// TIA Portal V16 export
// export: Created 2021-08-16T21:06:41.371237Z, ExportSetting WithDefaults, DisplayName Totally Integrated Automation Portal, DisplayVersion V16, DisplayName TIA Portal Version Control Interface, DisplayVersion V16, DisplayName TIA Portal Openness, DisplayVersion V16, DisplayName STEP 7 Professional, DisplayVersion V16, DisplayName STEP 7 Safety, DisplayVersion V16, DisplayName WinCC Advanced, DisplayVersion V16
ORGANIZATION_BLOCK "Main"   // OB1, LAD, ProgramCycle
TITLE = "Main Program Sweep (Cycle)"
{ S7_Optimized_Access := 'TRUE' }
VERSION : 0.1
// stored: AutoNumber true, IsIECCheckEnabled false, SetENOAutomatically false
   VAR_INPUT
      Initial_Call : Bool;   // Initial call of this OB
      Remanence : Bool;   // =True, if remanent data are available
   END_VAR
   VAR CONSTANT
      start : Bool;
   END_VAR
BEGIN

REGION Network 1: Spustenie a zastavenie automatického režimu
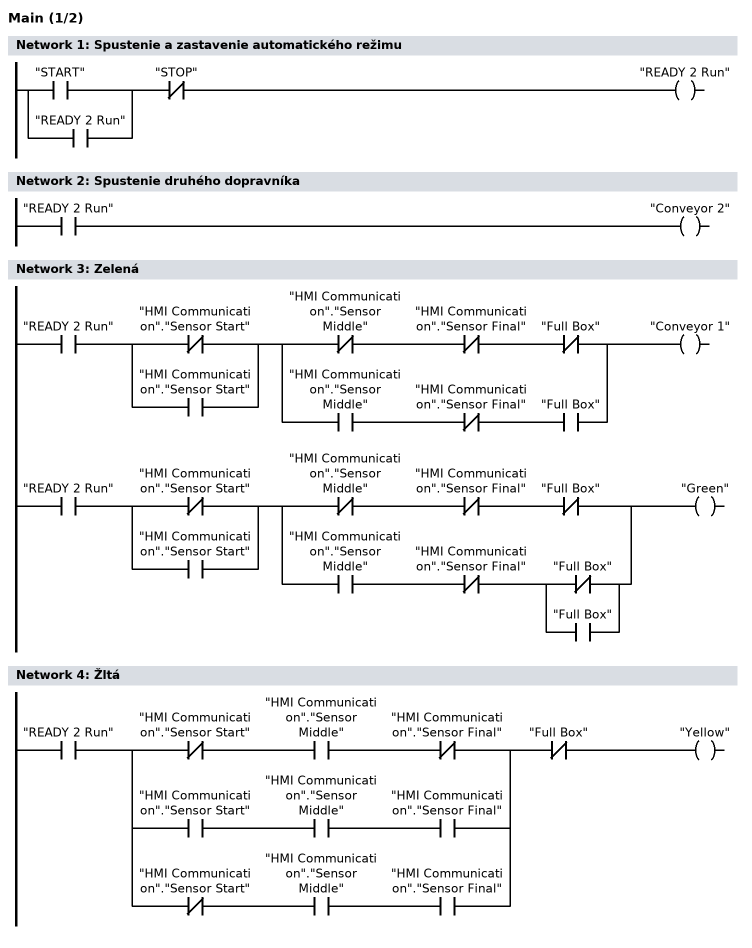
   RUNG wire#powerrail
      Contact( "START" )
      wire#w1
      I_Contact( "STOP" )
      Coil( "READY 2 Run" )
   END_RUNG
   RUNG wire#powerrail
      Contact( "READY 2 Run" )
   END_RUNG wire#w1
   // the same network as SCL:
   "READY 2 Run" := ("START" OR "READY 2 Run") AND NOT "STOP";
END_REGION

REGION Network 2: Spustenie druhého dopravníka
   RUNG wire#powerrail
      Contact( "READY 2 Run" )
      Coil( "Conveyor 2" )
   END_RUNG
   // the same network as SCL:
   "Conveyor 2" := "READY 2 Run";
END_REGION

REGION Network 3: Zelená
   RUNG wire#powerrail
      Contact( "READY 2 Run" )
      wire#w1
      I_Contact( "HMI Communication"."Sensor Start" )
      wire#w2
      I_Contact( "HMI Communication"."Sensor Middle" )
      I_Contact( "HMI Communication"."Sensor Final" )
      I_Contact( "Full Box" )
      wire#w3
      Coil( "Conveyor 1" )
   END_RUNG
   RUNG wire#w1
      Contact( "HMI Communication"."Sensor Start" )
   END_RUNG wire#w2
   RUNG wire#w2
      Contact( "HMI Communication"."Sensor Middle" )
      I_Contact( "HMI Communication"."Sensor Final" )
      Contact( "Full Box" )
   END_RUNG wire#w3
   RUNG wire#powerrail
      Contact( "READY 2 Run" )
      wire#w4
      I_Contact( "HMI Communication"."Sensor Start" )
      wire#w5
      I_Contact( "HMI Communication"."Sensor Middle" )
      I_Contact( "HMI Communication"."Sensor Final" )
      I_Contact( "Full Box" )
      wire#w6
      Coil( "Green" )
   END_RUNG
   RUNG wire#w4
      Contact( "HMI Communication"."Sensor Start" )
   END_RUNG wire#w5
   RUNG wire#w5
      Contact( "HMI Communication"."Sensor Middle" )
      I_Contact( "HMI Communication"."Sensor Final" )
      wire#w7
      I_Contact( "Full Box" )
   END_RUNG wire#w6
   RUNG wire#w7
      Contact( "Full Box" )
   END_RUNG wire#w6
   // the same network as SCL:
   "Conveyor 1" := "READY 2 Run" AND (NOT "HMI Communication"."Sensor Start" OR "HMI Communication"."Sensor Start") AND ((NOT "HMI Communication"."Sensor Middle" AND NOT "HMI Communication"."Sensor Final" AND NOT "Full Box") OR ("HMI Communication"."Sensor Middle" AND NOT "HMI Communication"."Sensor Final" AND "Full Box"));
   "Green" := "READY 2 Run" AND (NOT "HMI Communication"."Sensor Start" OR "HMI Communication"."Sensor Start") AND ((NOT "HMI Communication"."Sensor Middle" AND NOT "HMI Communication"."Sensor Final" AND NOT "Full Box") OR ("HMI Communication"."Sensor Middle" AND NOT "HMI Communication"."Sensor Final" AND (NOT "Full Box" OR "Full Box")));
END_REGION

REGION Network 4: Žltá
   RUNG wire#powerrail
      Contact( "READY 2 Run" )
      wire#w1
      I_Contact( "HMI Communication"."Sensor Start" )
      Contact( "HMI Communication"."Sensor Middle" )
      I_Contact( "HMI Communication"."Sensor Final" )
      wire#w2
      I_Contact( "Full Box" )
      Coil( "Yellow" )
   END_RUNG
   RUNG wire#w1
      Contact( "HMI Communication"."Sensor Start" )
      Contact( "HMI Communication"."Sensor Middle" )
      Contact( "HMI Communication"."Sensor Final" )
   END_RUNG wire#w2
   RUNG wire#w1
      I_Contact( "HMI Communication"."Sensor Start" )
      Contact( "HMI Communication"."Sensor Middle" )
      Contact( "HMI Communication"."Sensor Final" )
   END_RUNG wire#w2
   // the same network as SCL:
   "Yellow" := "READY 2 Run" AND ((NOT "HMI Communication"."Sensor Start" AND "HMI Communication"."Sensor Middle" AND NOT "HMI Communication"."Sensor Final") OR ("HMI Communication"."Sensor Start" AND "HMI Communication"."Sensor Middle" AND "HMI Communication"."Sensor Final") OR (NOT "HMI Communication"."Sensor Start" AND "HMI Communication"."Sensor Middle" AND "HMI Communication"."Sensor Final")) AND NOT "Full Box";
END_REGION

REGION Network 5: Červená
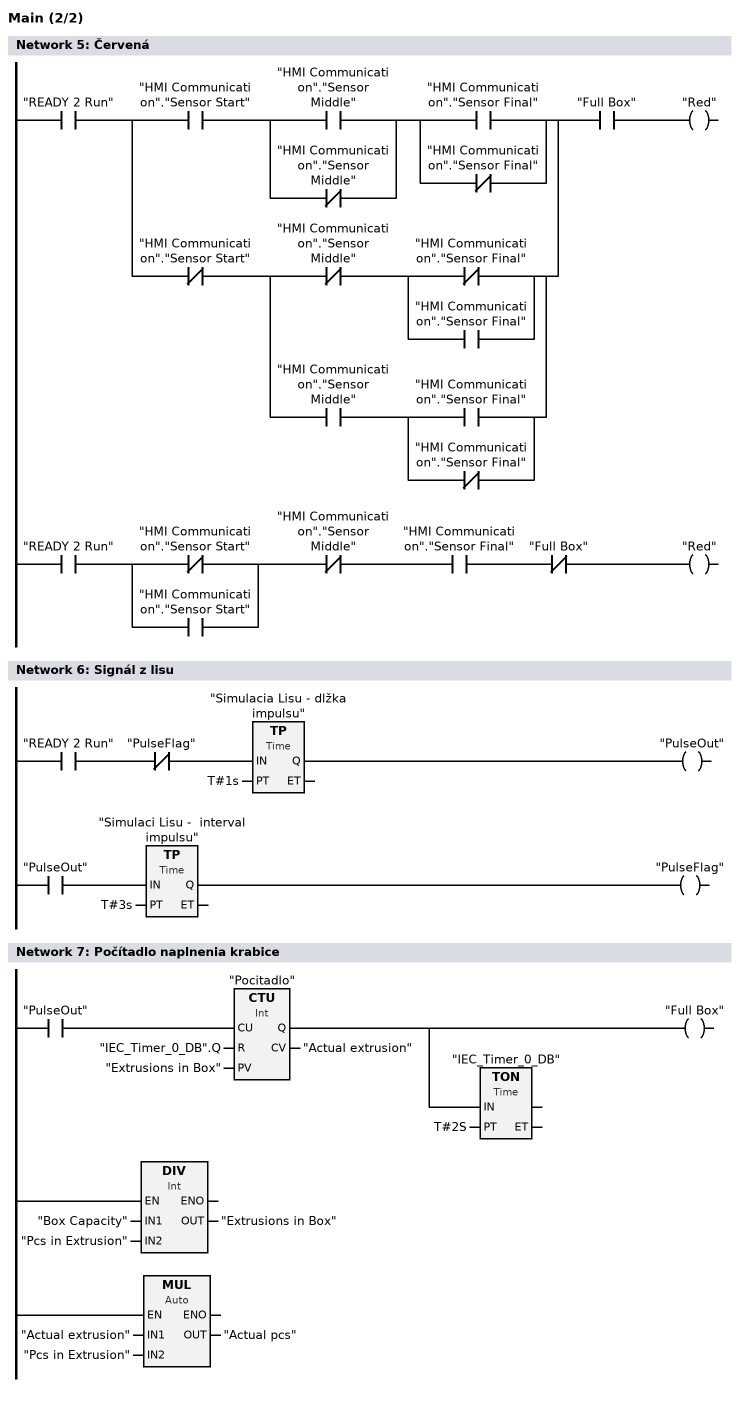
   RUNG wire#powerrail
      Contact( "READY 2 Run" )
      wire#w1
      Contact( "HMI Communication"."Sensor Start" )
      wire#w2
      Contact( "HMI Communication"."Sensor Middle" )
      wire#w3
      Contact( "HMI Communication"."Sensor Final" )
      wire#w4
      Contact( "Full Box" )
      Coil( "Red" )
   END_RUNG
   RUNG wire#w2
      I_Contact( "HMI Communication"."Sensor Middle" )
   END_RUNG wire#w3
   RUNG wire#w3
      I_Contact( "HMI Communication"."Sensor Final" )
   END_RUNG wire#w4
   RUNG wire#w1
      I_Contact( "HMI Communication"."Sensor Start" )
      wire#w5
      I_Contact( "HMI Communication"."Sensor Middle" )
      wire#w6
      I_Contact( "HMI Communication"."Sensor Final" )
   END_RUNG wire#w4
   RUNG wire#w6
      Contact( "HMI Communication"."Sensor Final" )
   END_RUNG wire#w4
   RUNG wire#w5
      Contact( "HMI Communication"."Sensor Middle" )
      wire#w7
      Contact( "HMI Communication"."Sensor Final" )
   END_RUNG wire#w4
   RUNG wire#w7
      I_Contact( "HMI Communication"."Sensor Final" )
   END_RUNG wire#w4
   RUNG wire#powerrail
      Contact( "READY 2 Run" )
      wire#w8
      I_Contact( "HMI Communication"."Sensor Start" )
      wire#w9
      I_Contact( "HMI Communication"."Sensor Middle" )
      Contact( "HMI Communication"."Sensor Final" )
      I_Contact( "Full Box" )
      Coil( "Red" )
   END_RUNG
   RUNG wire#w8
      Contact( "HMI Communication"."Sensor Start" )
   END_RUNG wire#w9
   // the same network as SCL:
   "Red" := "READY 2 Run" AND (("HMI Communication"."Sensor Start" AND ("HMI Communication"."Sensor Middle" OR NOT "HMI Communication"."Sensor Middle") AND ("HMI Communication"."Sensor Final" OR NOT "HMI Communication"."Sensor Final")) OR (NOT "HMI Communication"."Sensor Start" AND ((NOT "HMI Communication"."Sensor Middle" AND (NOT "HMI Communication"."Sensor Final" OR "HMI Communication"."Sensor Final")) OR ("HMI Communication"."Sensor Middle" AND ("HMI Communication"."Sensor Final" OR NOT "HMI Communication"."Sensor Final"))))) AND "Full Box";
   "Red" := "READY 2 Run" AND (NOT "HMI Communication"."Sensor Start" OR "HMI Communication"."Sensor Start") AND NOT "HMI Communication"."Sensor Middle" AND "HMI Communication"."Sensor Final" AND NOT "Full Box";
END_REGION

REGION Network 6: Signál z lisu
   RUNG wire#powerrail
      Contact( "READY 2 Run" )
      I_Contact( "PulseFlag" )
      { S7_Templates := "time_type := Time" } "Simulacia Lisu - dlžka impulsu".TP(pt := T#1s, et =>)
      Coil( "PulseOut" )
   END_RUNG
   RUNG wire#powerrail
      Contact( "PulseOut" )
      { S7_Templates := "time_type := Time" } "Simulaci Lisu -  interval impulsu".TP(pt := T#3s, et =>)
      Coil( "PulseFlag" )
   END_RUNG
   // the same network as SCL:
   "Simulacia Lisu - dlžka impulsu".TP(IN := "READY 2 Run" AND NOT "PulseFlag", PT := T#1s);
   "PulseOut" := "Simulacia Lisu - dlžka impulsu".Q;
   "Simulaci Lisu -  interval impulsu".TP(IN := "PulseOut", PT := T#3s);
   "PulseFlag" := "Simulaci Lisu -  interval impulsu".Q;
END_REGION

REGION Network 7: Počítadlo naplnenia krabice
   RUNG wire#powerrail
      Contact( "PulseOut" )
      { S7_Templates := "value_type := Int" } "Pocitadlo".CTU(r := "IEC_Timer_0_DB".Q, pv := "Extrusions in Box", cv => "Actual extrusion")
      wire#w1
      Coil( "Full Box" )
   END_RUNG
   RUNG wire#w1
      { S7_Templates := "time_type := Time" } "IEC_Timer_0_DB".TON(pt := T#2S, et =>)
   END_RUNG
   RUNG wire#powerrail
      { S7_Templates := "SrcType := Int" } Div(in1 := "Box Capacity", in2 := "Pcs in Extrusion", out => "Extrusions in Box")
   END_RUNG
   RUNG wire#powerrail
      Mul(in1 := "Actual extrusion", in2 := "Pcs in Extrusion", out => "Actual pcs")
   END_RUNG
   // the same network as SCL:
   "Pocitadlo".CTU(CU := "PulseOut",
                   R := "IEC_Timer_0_DB".Q,
                   PV := "Extrusions in Box",
                   CV => "Actual extrusion");
   "Full Box" := "Pocitadlo".Q;
   "IEC_Timer_0_DB".TON(IN := "Pocitadlo".Q, PT := T#2S);
   "Extrusions in Box" := "Box Capacity" / "Pcs in Extrusion";
   "Actual pcs" := "Actual extrusion" * "Pcs in Extrusion";
END_REGION
END_ORGANIZATION_BLOCK
